// Mitsubishi GX Works2 project: AI机程序250116-动作串联运行准备   PLC: FX3S

PROGRAM MAIN
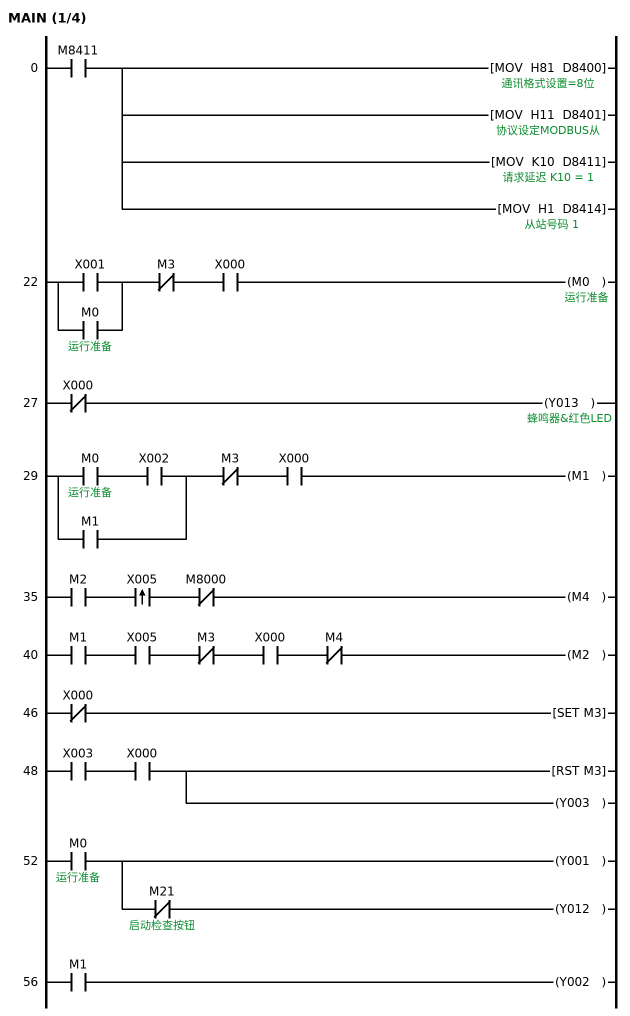
0     LD      M8411
      MOV     H81 D8400  ; 通讯格式设置=8位
      MOV     H11 D8401  ; 协议设定MODBUS从
      MOV     K10 D8411  ; 请求延迟 K10 = 1
      MOV     H1 D8414  ; 从站号码 1
22    LD      X001
      OR      M0  ; 运行准备
      ANI     M3
      AND     X000
      OUT     M0  ; 运行准备
27    LDI     X000
      OUT     Y013  ; 蜂鸣器&红色LED
29    LD      M0  ; 运行准备
      AND     X002
      OR      M1
      ANI     M3
      AND     X000
      OUT     M1
35    LD      M2
      ANDP    X005
      ANI     M8000
      OUT     M4
40    LD      M1
      AND     X005
      ANI     M3
      AND     X000
      ANI     M4
      OUT     M2
46    LDI     X000
      SET     M3
48    LD      X003
      AND     X000
      RST     M3
      OUT     Y003
52    LD      M0  ; 运行准备
      OUT     Y001
      ANI     M21  ; 启动检查按钮
      OUT     Y012
56    LD      M1
      OUT     Y002
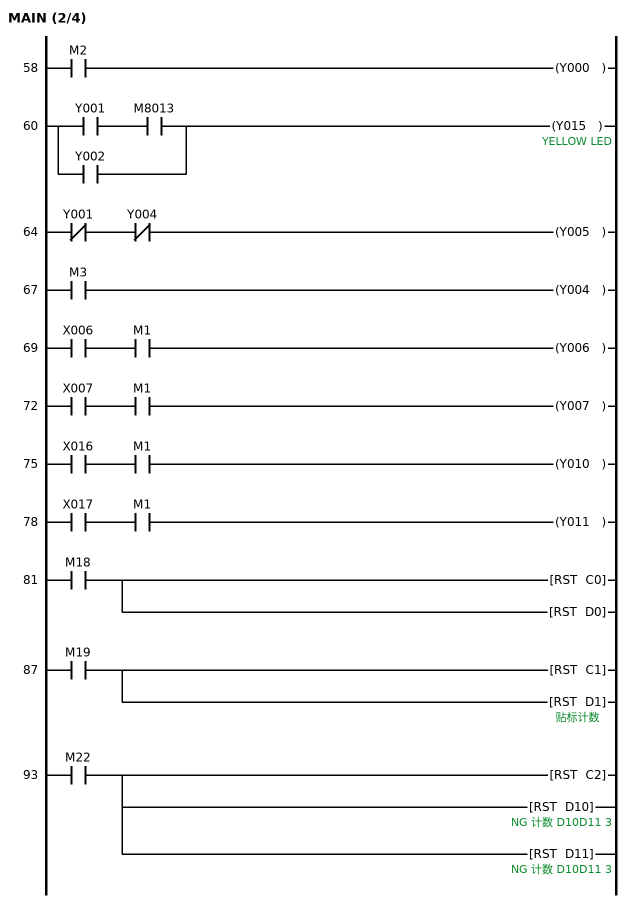
58    LD      M2
      OUT     Y000
60    LD      Y001
      AND     M8013
      OR      Y002
      OUT     Y015  ; YELLOW LED
64    LDI     Y001
      ANI     Y004
      OUT     Y005
67    LD      M3
      OUT     Y004
69    LD      X006
      AND     M1
      OUT     Y006
72    LD      X007
      AND     M1
      OUT     Y007
75    LD      X016
      AND     M1
      OUT     Y010
78    LD      X017
      AND     M1
      OUT     Y011
81    LD      M18
      RST     C0
      RST     D0
87    LD      M19
      RST     C1
      RST     D1  ; 贴标计数
93    LD      M22
      RST     C2
      RST     D10  ; NG 计数 D10D11 3
      RST     D11  ; NG 计数 D10D11 3
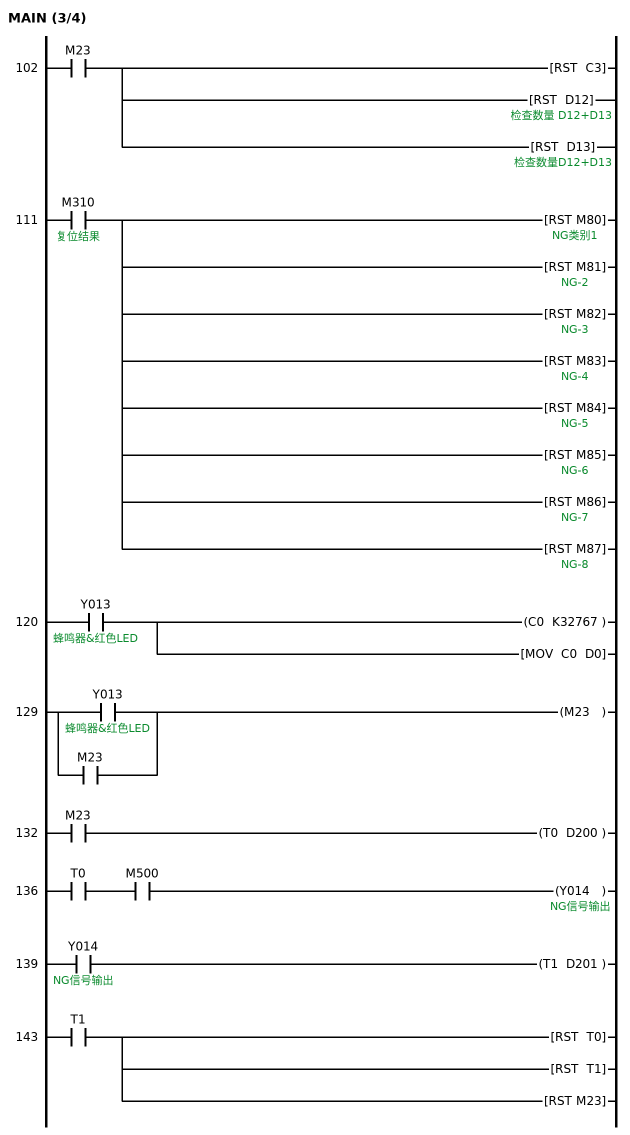
102   LD      M23
      RST     C3
      RST     D12  ; 检查数量 D12+D13
      RST     D13  ; 检查数量D12+D13
111   LD      M310  ; 复位结果
      RST     M80  ; NG类别1
      RST     M81  ; NG-2
      RST     M82  ; NG-3
      RST     M83  ; NG-4
      RST     M84  ; NG-5
      RST     M85  ; NG-6
      RST     M86  ; NG-7
      RST     M87  ; NG-8
120   LD      Y013  ; 蜂鸣器&红色LED
      OUT     C0 K32767
      MOV     C0 D0
129   LD      Y013  ; 蜂鸣器&红色LED
      OR      M23
      OUT     M23
132   LD      M23
      OUT     T0 D200
136   LD      T0
      AND     M500
      OUT     Y014  ; NG信号输出
139   LD      Y014  ; NG信号输出
      OUT     T1 D201
143   LD      T1
      RST     T0
      RST     T1
      RST     M23
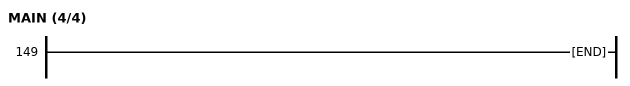
149   END
END_PROGRAM

// device comments not shown above
M300  ; 控制开关-GOT
M520  ; NG时输出有效
